PROGRAM Ax_01_AxisIncrementSelect_04
VAR
	HMI_Motion: FB_HMI_Control;


	tMessageOffset: UINT;
	tNumMessagesPerRow: UINT;
	
	
	MyAdvanceInterlock: BOOL;
	MyReturnInterlock: BOOL;
	
	MyAutoAdvanceCondition: BOOL;
	MyAutoReturnCondition: BOOL;
	
	myAdvancePrompt: BOOL;
	myReturnPrompt: BOOL;
	

	NotUsed: UINT;
	
	selection :INT;
	

END_VAR
VAR // added by the converter: edge detectors and wires of the graphical bodies
    _w1 : BOOL;
    _rt1, _rt2 : R_TRIG;
END_VAR

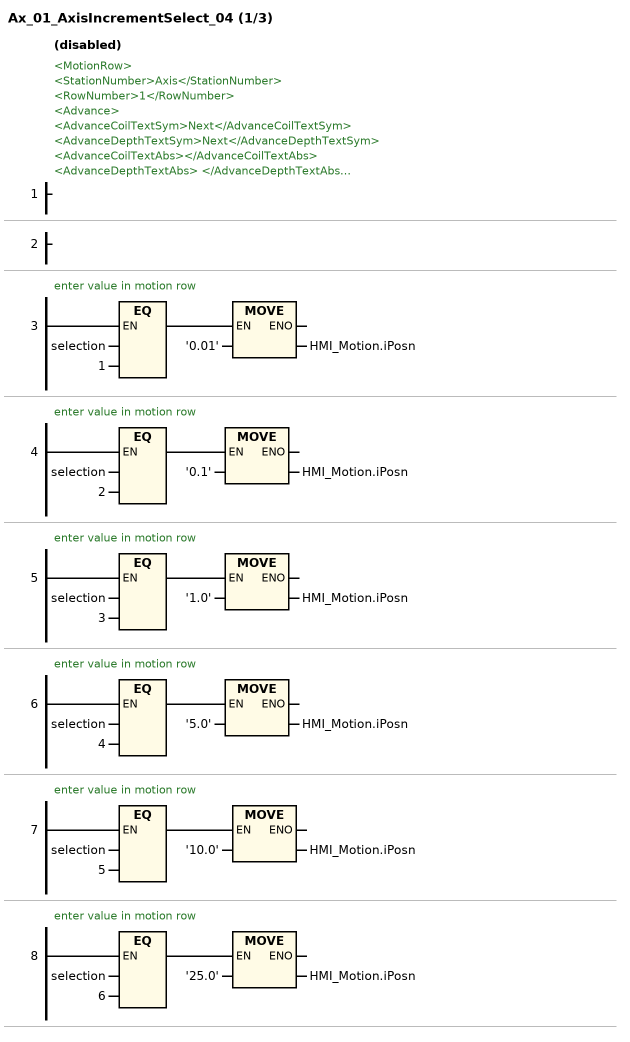
// NETWORK 1 (disabled)
// <MotionRow>
// <StationNumber>Axis</StationNumber>
// <RowNumber>1</RowNumber>
//   <Advance>
//     <AdvanceCoilTextSym>Next</AdvanceCoilTextSym>
//     <AdvanceDepthTextSym>Next</AdvanceDepthTextSym>
//     <AdvanceCoilTextAbs></AdvanceCoilTextAbs>
//     <AdvanceDepthTextAbs> </AdvanceDepthTextAbs>
//     <ManSeq></ManSeq>
//   </Advance>
//   <Return>
//     <ReturnCoilTextSym>Previous</ReturnCoilTextSym>
//     <ReturnDepthTextSym>Previous</ReturnDepthTextSym>
//     <ReturnCoilTextAbs></ReturnCoilTextAbs>
//     <ReturnDepthTextAbs></ReturnDepthTextAbs>
//    <ManSeq></ManSeq>
//   </Return>
//   <Motion>
//     <NameSym>Axis Name</NameSym>
//     <NameAbs>X1</NameAbs>
//   </Motion>
// </MotionRow>

// NETWORK 2

// NETWORK 3
// enter value in motion row
IF selection = 1 THEN HMI_Motion.iPosn := '0.01'; END_IF

// NETWORK 4
// enter value in motion row
IF selection = 2 THEN HMI_Motion.iPosn := '0.1'; END_IF

// NETWORK 5
// enter value in motion row
IF selection = 3 THEN HMI_Motion.iPosn := '1.0'; END_IF

// NETWORK 6
// enter value in motion row
IF selection = 4 THEN HMI_Motion.iPosn := '5.0'; END_IF

// NETWORK 7
// enter value in motion row
IF selection = 5 THEN HMI_Motion.iPosn := '10.0'; END_IF

// NETWORK 8
// enter value in motion row
IF selection = 6 THEN HMI_Motion.iPosn := '25.0'; END_IF

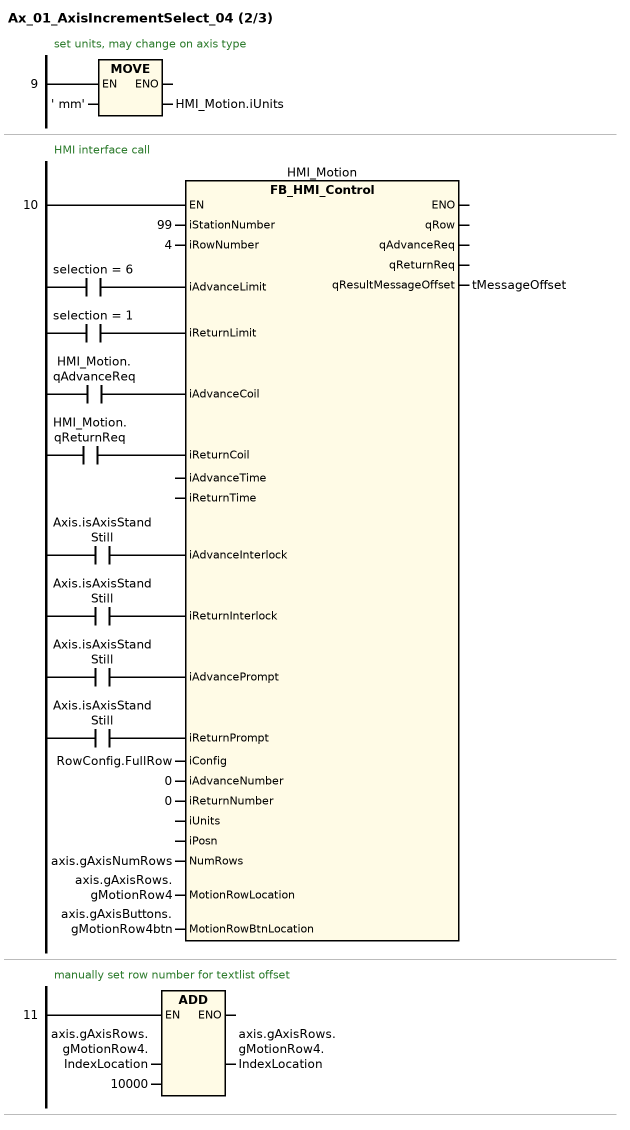
// NETWORK 9
// set units, may change on axis type
HMI_Motion.iUnits := ' mm';

// NETWORK 10
// HMI interface call
HMI_Motion(
    iStationNumber := 99,
    iRowNumber := 4,
    iAdvanceLimit := selection = 6,
    iReturnLimit := selection = 1,
    iAdvanceCoil := HMI_Motion.qAdvanceReq,
    iReturnCoil := HMI_Motion.qReturnReq,
    iAdvanceInterlock := Axis.isAxisStandStill,
    iReturnInterlock := Axis.isAxisStandStill,
    iAdvancePrompt := Axis.isAxisStandStill,
    iReturnPrompt := Axis.isAxisStandStill,
    iConfig := RowConfig.FullRow,
    iAdvanceNumber := 0,
    iReturnNumber := 0,
    NumRows := axis.gAxisNumRows,
    MotionRowLocation := axis.gAxisRows.gMotionRow4,
    MotionRowBtnLocation := axis.gAxisButtons.gMotionRow4btn,
    qResultMessageOffset => tMessageOffset); // FB_HMI_Control

// NETWORK 11
// manually set row number for textlist offset
axis.gAxisRows.gMotionRow4.IndexLocation := axis.gAxisRows.gMotionRow4.IndexLocation + 10000;

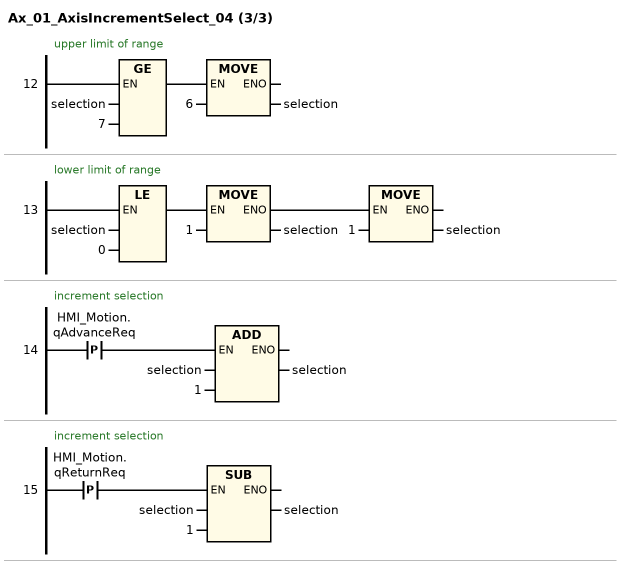
// NETWORK 12
// upper limit of range
IF selection >= 7 THEN selection := 6; END_IF

// NETWORK 13
// lower limit of range
_w1 := selection <= 0;
IF _w1 THEN selection := 1; END_IF
IF _w1 THEN selection := 1; END_IF

// NETWORK 14
// increment selection
_rt1(CLK := HMI_Motion.qAdvanceReq);
IF _rt1.Q THEN selection := selection + 1; END_IF

// NETWORK 15
// increment selection
_rt2(CLK := HMI_Motion.qReturnReq);
IF _rt2.Q THEN selection := selection - 1; END_IF

END_PROGRAM

(* stored: Version 1.1.0.1, ProductVersion 3.1.4024.12
   POU Ax_01_AxisIncrementSelect_04: Id {8ba27c82-4140-4ab7-a605-a25b71940dcc}, SpecialFunc None *)
